% RSLogix 500 project PROJECT8.RSS, saved by version 8.40.00.08 %
PROJECT "UNTITLED"    % processor: Bul.1763 MicroLogix 1100 Series B %

PROGRAM FILES
  LAD 2   12 rungs

DATA FILES
  O0 OUTPUT  4 elements
  I1 INPUT  6 elements
  S2 STATUS  66 elements
  B3 BINARY  1 elements
  T4 TIMER  1 elements
  C5 COUNTER  1 elements
  R6 CONTROL  1 elements
  N7 INTEGER  4 elements
  F8 FLOAT  3 elements

LADDER 2
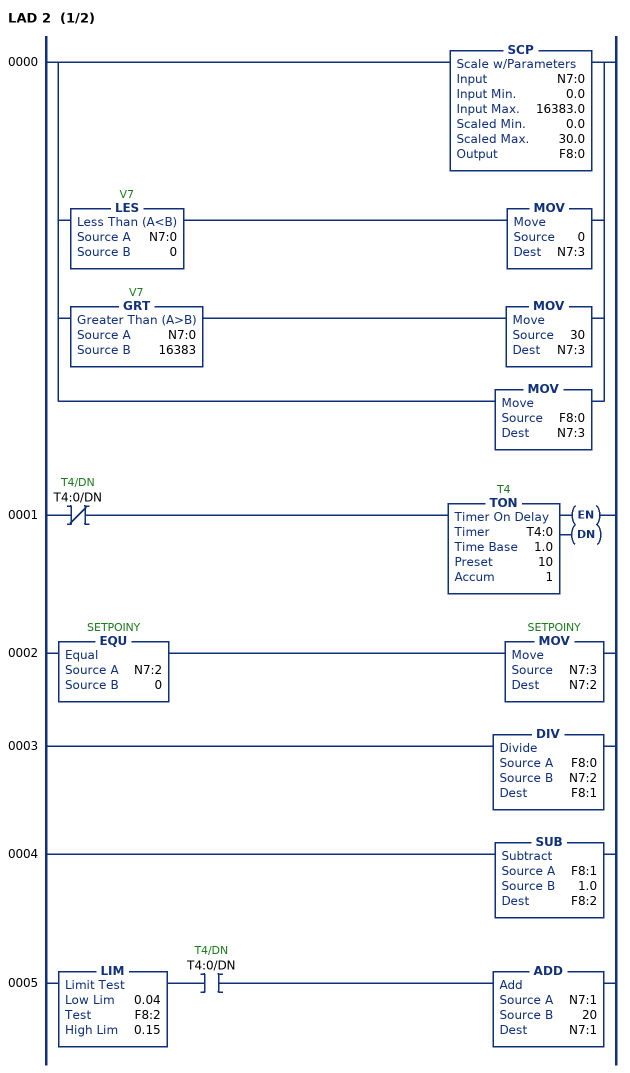
% Rung: 0 %
SOR BST SCP N7:0 0.0 16383.0 0.0 30.0 F8:0 NXB LES N7:0 0 MOV 0 N7:3 NXB GRT N7:0 16383 MOV 30 N7:3 NXB MOV F8:0 N7:3 BND EOR
%   N7:0  V7 %
% Rung: 1 %
SOR XIO T4:0/DN TON T4:0 1.0 10 1 EOR
%   T4:0  T4 %
% Rung: 2 %
SOR EQU N7:2 0 MOV N7:3 N7:2 EOR
%   N7:2  SETPOINY %
% Rung: 3 %
SOR DIV F8:0 N7:2 F8:1 EOR
%   N7:2  SETPOINY %
% Rung: 4 %
SOR SUB F8:1 1.0 F8:2 EOR
% Rung: 5 %
SOR LIM 0.04 F8:2 0.15 XIC T4:0/DN ADD N7:1 20 N7:1 EOR
%   T4:0  T4 %

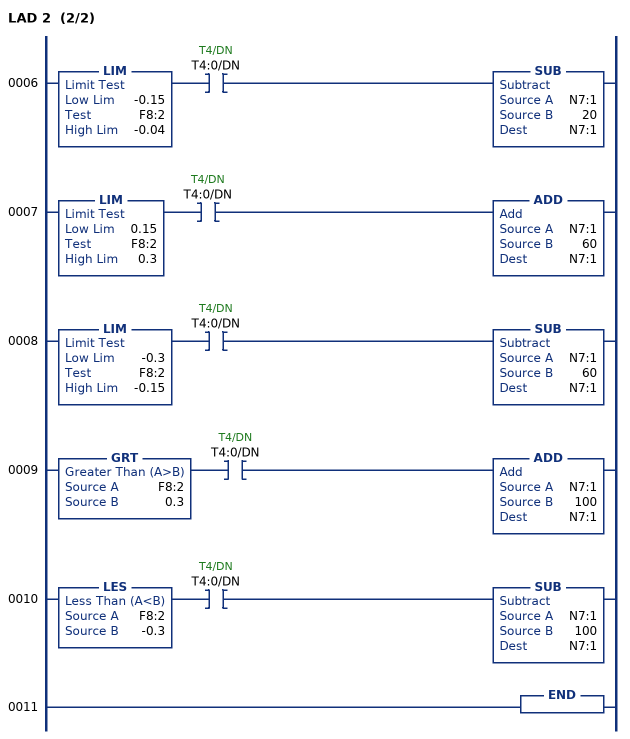
% Rung: 6 %
SOR LIM -0.15 F8:2 -0.04 XIC T4:0/DN SUB N7:1 20 N7:1 EOR
%   T4:0  T4 %
% Rung: 7 %
SOR LIM 0.15 F8:2 0.3 XIC T4:0/DN ADD N7:1 60 N7:1 EOR
%   T4:0  T4 %
% Rung: 8 %
SOR LIM -0.3 F8:2 -0.15 XIC T4:0/DN SUB N7:1 60 N7:1 EOR
%   T4:0  T4 %
% Rung: 9 %
SOR GRT F8:2 0.3 XIC T4:0/DN ADD N7:1 100 N7:1 EOR
%   T4:0  T4 %
% Rung: 10 %
SOR LES F8:2 -0.3 XIC T4:0/DN SUB N7:1 100 N7:1 EOR
%   T4:0  T4 %
% Rung: 11 %
SOR END EOR

DATA TABLE (non-zero values as saved)
DATA T4
% .PRE .ACC %
% T4:0 % 10 1
DATA N7
% N7:0 % 8192 6020 15 15
DATA F8
% F8:0 % 15.00092 1.000061 6.103516e-05
